Universal Robots PolyScope program: ferranmarinaP1.urp

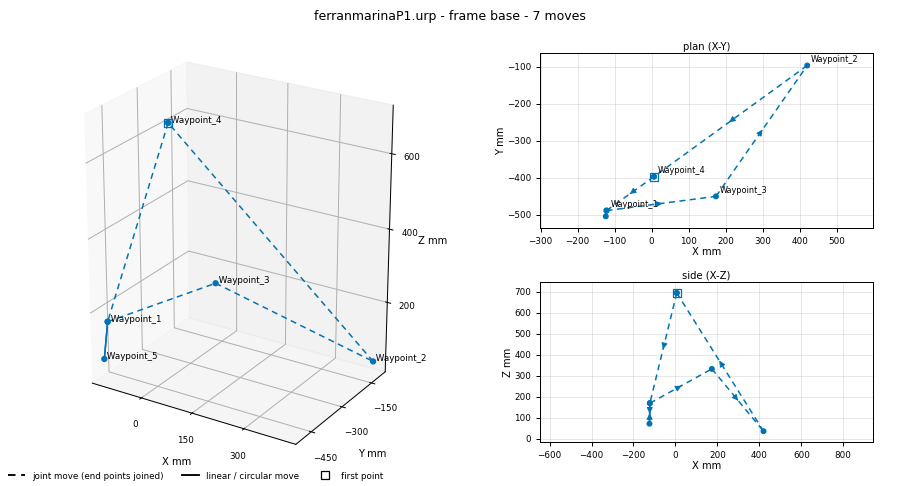
[picture p0: tool path of ferranmarinaP1.urp in frame base, 7 of 7 moves have a stored position in this frame; points joined in program order, loops and branches not executed]
Program ferranmarinaP1 (installation=default directory=/programs createdIn=5.14.5 lastSavedIn=5.14.5 robotSerialNumber=20195300809)
Calibrated DH parameters: a=[-0.000085, -0.20076, -0.212369, 0.000121, -0.000118, 0]; d=[0.15185, -26.306375, 24.753047, 1.684739, 0.085386, 0.092088]; alpha=[1.572149, -0.00522, -0.011864, 1.571339, -1.571085, 0]; deltaTheta=[0, 0.599885, -0.513355, -0.086555, 0.000006, 0]
InitVariablesNode
Robot Program (runOnlyOnce=false)
  MoveJ speed 60 deg/s, acceleration 80 deg/s^2 (useActiveTCP=true) feature=Base
    Waypoint Waypoint_4: TCP in base x=6.312 y=-396.697 z=694.741 mm, rx=-0.0179 ry=2.2101 rz=-2.2165 rad; joints [-0.001, -89.998, 0.001, -90.001, 0.002, 0] deg; TCP offset x=0 y=0 z=174 mm, rx=0 ry=0 rz=0 rad
  Set DigitalOutput pin=digital_out[0]; digitalValue=1
  MoveJ speed 60 deg/s, acceleration 80 deg/s^2 (useActiveTCP=true) feature=Base
    Waypoint Waypoint_1: TCP in base x=-121.854 y=-488.305 z=169.423 mm, rx=0.0545 ry=-3.1094 rz=0.2104 rad; joints [-88.248, -150.24, 15.085, -127.127, 87.746, 0.368] deg
  Wait DigitalInput pin=digital_in[0]; digitalValue=0
  Set DigitalOutput pin=digital_out[0]; digitalValue=0
  MoveL speed 250 mm/s, acceleration 1200 mm/s^2 (useActiveTCP=true) feature=Base
    Waypoint Waypoint_5: TCP in base x=-123.854 y=-503.95 z=71.615 mm, rx=0.0047 ry=-3.1159 rz=-0.0093 rad; joints [-88.581, -155.662, 0.004, -114.72, 87.715, 1.877] deg
    URCap Gripper (Robotiq_Grippers, Robotiq Inc.) dataModel(position=56.3921568627451, force=0.0, speed=0.0, positionInDouble=56.3921568627451, forceInDouble=0.0, speedInDouble=0.0, slaveIds=[9], blocking=true)
    Waypoint Waypoint_1: TCP in base x=-121.854 y=-488.305 z=169.423 mm, rx=0.0545 ry=-3.1094 rz=0.2104 rad; joints [-88.248, -150.24, 15.085, -127.127, 87.746, 0.368] deg
  Set DigitalOutput pin=digital_out[0]; digitalValue=1
  MoveJ speed 60 deg/s, acceleration 80 deg/s^2 (useActiveTCP=true) feature=Base
    Waypoint Waypoint_3: motionParameters(blendRadius=0.05); TCP in base x=173.537 y=-450.009 z=332.692 mm, rx=-0.95 ry=2.7044 rz=-0.7268 rad; joints [-54.65, -115.944, -19.422, -104.362, 91.518, -2.233] deg
  If cont>3
    Wait Sleep waitTime=20
    cont := 0
  MoveJ speed 60 deg/s, acceleration 80 deg/s^2 (useActiveTCP=true) feature=Base
    Waypoint Waypoint_2: TCP in base x=419.908 y=-96.836 z=35.768 mm, rx=2.2122 ry=-2.1785 rz=-0.0844 rad; joints [3.874, -123.79, -68.61, -81.173, 90.24, 3.254] deg
    URCap Gripper Activate (Robotiq_Grippers, Robotiq Inc.) dataModel(ResetAndActivateKey=false)
    URCap Gripper (Robotiq_Grippers, Robotiq Inc.) dataModel(position=0.0, force=0.0, speed=0.0, positionInDouble=0.0, forceInDouble=0.0, speedInDouble=0.0, slaveIds=[9], blocking=true)
    Waypoint Waypoint_4: TCP in base x=6.312 y=-396.697 z=694.741 mm, rx=-0.0179 ry=2.2101 rz=-2.2165 rad; joints [-0.001, -89.998, 0.001, -90.001, 0.002, 0] deg
  cont := cont+1
